FUNCTION_BLOCK FB_SimulatedOutOpen_DG IMPLEMENTS ITF_Regelschuif_OutOpen_DG
VAR
	internalState : BOOL := FALSE;
END_VAR

METHOD set : BOOL
VAR_INPUT
	state : BOOL;
END_VAR
internalState := state;
END_METHOD

END_FUNCTION_BLOCK

(* stored: Version 1.1.0.1, ProductVersion 3.1.4026.8
   POU FB_SimulatedOutOpen_DG: Id {dd7eec1a-cd3e-4e90-b599-3cbc509f8f0e}, SpecialFunc None
   Method set: Id {832fdc31-444b-4857-8ebe-29836373b23b} *)
